(* CODESYS project Untitled1.project

Project tree, tasks and I/O mapping:
  Device : CECC-S, Festo AG & Co. KG, order no. 574416, version 3.5.4.0
    application Application
      libraries: Standard, * (System)
      task MainTask (cyclic, interval t#20ms, priority 20) calls PLC_PRG
      program PLC_PRG [ST]
    Onboard : CECC 14I/8O, Festo AG & Co. KG, version 3.4.5.5
        unmapped channels: Onboard Input, Onboard Output
      Digital Inputs
          unmapped channels: Onboard Input
      Digital Outputs
          unmapped channels: Onboard Output
*)

// Device/Application/PLC_PRG
PROGRAM PLC_PRG
VAR Hello:BOOL;
	Brett:BOOL;
	Version2:bool;
END_VAR

Hello;

Brett;

Version2;

END_PROGRAM
